INTERFACE ITF_PackMLState

METHOD CyclicLogic : BOOL
VAR_INPUT
END_VAR
END_METHOD

METHOD EStop : BOOL
VAR_INPUT
END_VAR
END_METHOD

METHOD Reset : BOOL
VAR_INPUT
END_VAR
END_METHOD

METHOD SetContext : BOOL
VAR_INPUT
	context : ITF_PackMLMachine;
END_VAR
END_METHOD

METHOD Start : BOOL
VAR_INPUT
END_VAR
END_METHOD

METHOD Stop : BOOL
VAR_INPUT
END_VAR
END_METHOD

END_INTERFACE

(* stored: Version 1.1.0.1, ProductVersion 3.1.4024.12
   Itf ITF_PackMLState: Id {e9c1366e-6fde-42b1-a453-45ddf914b23a}
   Method CyclicLogic: Id {8098c19c-5131-4968-a6ba-edce4f338178}
   Method EStop: Id {02a9ba80-d1a4-4114-bdb6-ae917084a07b}
   Method Reset: Id {67e4205b-ea17-4b05-914c-cbb517da0b9f}
   Method SetContext: Id {64c80388-81c6-4c21-b859-370cc7ce1276}
   Method Start: Id {98d27ca1-d0a4-442e-867f-f84e49283cd4}
   Method Stop: Id {42ec46a1-995b-4534-977a-fa77637986f4} *)
